INTERFACE ITF_Component_TE1 EXTENDS ITF_BaseComponent

METHOD testMethod : BOOL
VAR_INPUT
END_VAR
END_METHOD

END_INTERFACE

(* stored: Version 1.1.0.1, ProductVersion 3.1.4024.15
   Itf ITF_Component_TE1: Id {502a6bad-580a-44ca-8c6b-64e750df33c8}
   Method testMethod: Id {1b12d73c-c685-4061-839e-c2f44dd24fd0} *)
